// TIA Portal V18 export
DATA_BLOCK "KeyenceSR1000Ctrl_803A1DB"   // DB1802
// stored: AutoNumber false, InstanceOfName KeyenceSR1000Ctrl, InstanceOfType FB
"KeyenceSR1000Ctrl"
   // VAR_INPUT
   //    iI_Address { ExternalAccessible := 'False'; ExternalVisible := 'False'; ExternalWritable := 'False'} : Int;
   //    iO_Address : Int;
   //    iSysRun : Bool;
   //    iReset : Bool;
   //    iAuto : Bool;
   //    iManual : Bool;
   //    iReTriggerLimitTimes : USInt;
   // END_VAR
   // VAR_OUTPUT
   //    oReady : Bool;
   //    oComplete : Bool;
   //    oError : Bool;
   //    oErrorCode : UInt;
   // END_VAR
   // VAR_IN_OUT
   //    ioAutoTrigger : Bool;
   // END_VAR
   // VAR
   //    sHMI { S7_SetPoint := 'True'} : "RCS_KeyenceSR1000_HMI";
   //    sCtrl : Struct
   //       Sequence : Int;
   //    END_STRUCT;
   //    sCurrentCode : String[128];
   //    sInData { S7_SetPoint := 'True'} : "RCS_KeyenceSR1000_Input";
   //    sOutData { S7_SetPoint := 'True'} : "RCS_KeyenceSR1000_Output";
   //    sAutoOld : Bool;
   //    sManualOld : Bool;
   //    sBusyTimeOut : Bool;
   //    sRunTimer { S7_SetPoint := 'True'} : TON_TIME;
   //    sBusyTimer { S7_SetPoint := 'True'} : TON_TIME;
   //    sFindCurrentPos { S7_SetPoint := 'True'} : Int;
   // END_VAR
BEGIN
END_DATA_BLOCK
